// TIA Portal V15.1 export
// export: Created 2020-06-12T07:35:47.5693359Z, ExportSetting None, DisplayName Totally Integrated Automation Portal, DisplayVersion V15.1, DisplayName TIA Portal Openness, DisplayVersion V15.1, DisplayName STEP 7 Professional, DisplayVersion V15.1, DisplayName STEP 7 Safety, DisplayVersion V15.1, DisplayName WinCC Advanced, DisplayVersion V15.1
FUNCTION "DED_Fan" : Void   // FC553, FBD
TITLE = Dedusting unit (SINK) control
{ S7_Optimized_Access := 'TRUE' }
// stored: SetENOAutomatically True
   VAR_TEMP
      tRelSpeed : Real;
      tFanSpeedMin : Real;
      tFanSpeedMax : Real;
      tActPress : Real;
      tClock : Bool;
      tDoSchake : Bool;
      tSpdContLock : Bool;
      tSetPress : Real;
   END_VAR
BEGIN

REGION Network 1: AX1LD3.M01: Fan
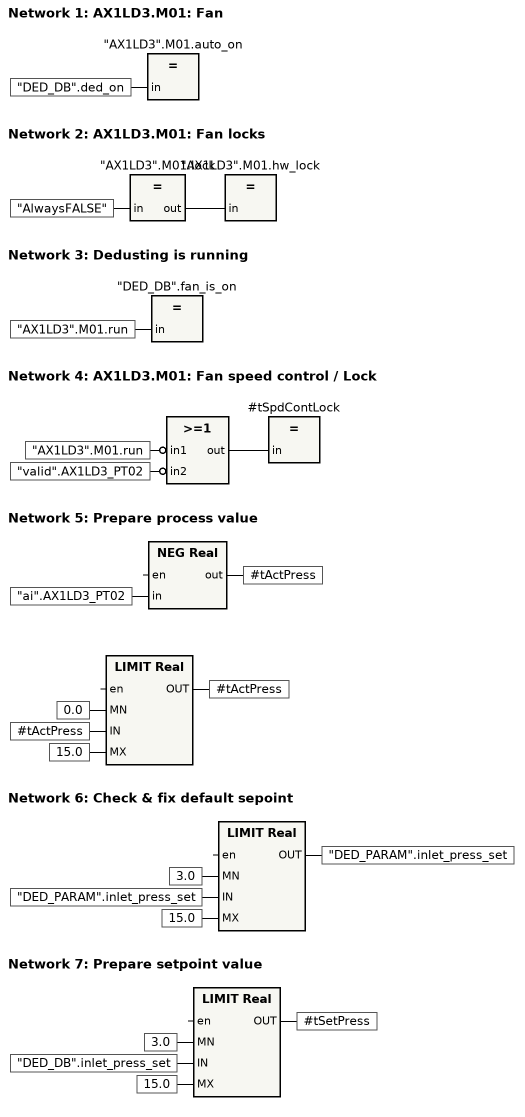
   "AX1LD3".M01.auto_on := "DED_DB".ded_on;
END_REGION

REGION Network 2: AX1LD3.M01: Fan locks
   "AX1LD3".M01.lock := "AlwaysFALSE";
   "AX1LD3".M01.hw_lock := "AlwaysFALSE";
END_REGION

REGION Network 3: Dedusting is running
   "DED_DB".fan_is_on := "AX1LD3".M01.run;
END_REGION

REGION Network 4: AX1LD3.M01: Fan speed control / Lock
   #tSpdContLock := NOT "AX1LD3".M01.run OR NOT "valid".AX1LD3_PT02;
END_REGION

REGION Network 5: Prepare process value
   #tActPress := -"ai".AX1LD3_PT02;
   #tActPress := LIMIT(MN := 0.0, IN := #tActPress, MX := 15.0);
END_REGION

REGION Network 6: Check & fix default sepoint
   "DED_PARAM".inlet_press_set := LIMIT(MN := 3.0, IN := "DED_PARAM".inlet_press_set, MX := 15.0);
END_REGION

REGION Network 7: Prepare setpoint value
   #tSetPress := LIMIT(MN := 3.0, IN := "DED_DB".inlet_press_set, MX := 15.0);
END_REGION

REGION Network 8: AX1LD3.M01: Fan speed control
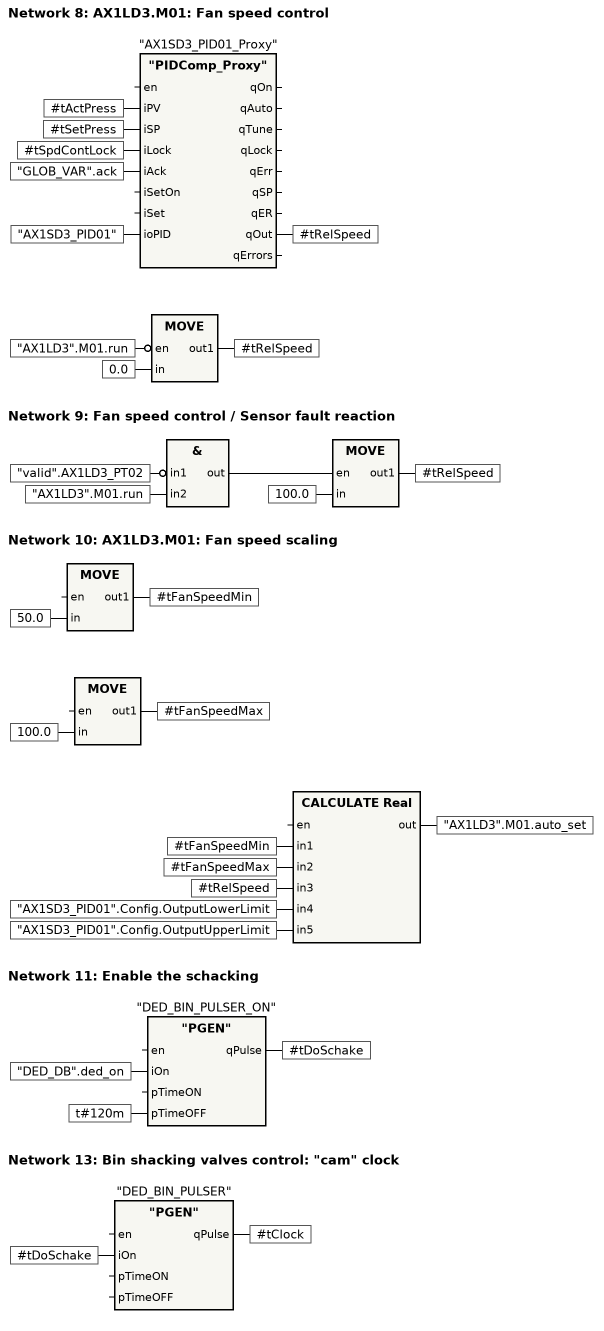
   "AX1SD3_PID01_Proxy"(iPV := #tActPress,   // "PIDComp_Proxy"
                        iSP := #tSetPress,
                        iLock := #tSpdContLock,
                        iAck := "GLOB_VAR".ack,
                        ioPID := "AX1SD3_PID01",
                        qOut => #tRelSpeed);
   IF NOT "AX1LD3".M01.run THEN #tRelSpeed := 0.0; END_IF;
END_REGION

REGION Network 9: Fan speed control / Sensor fault reaction
   IF NOT "valid".AX1LD3_PT02 AND "AX1LD3".M01.run THEN #tRelSpeed := 100.0; END_IF;
END_REGION

REGION Network 10: AX1LD3.M01: Fan speed scaling
   #tFanSpeedMin := 50.0;
   #tFanSpeedMax := 100.0;
   "AX1LD3".M01.auto_set := #tFanSpeedMin + (#tFanSpeedMax - #tFanSpeedMin) * ((#tRelSpeed - "AX1SD3_PID01".Config.OutputLowerLimit) / ("AX1SD3_PID01".Config.OutputUpperLimit - "AX1SD3_PID01".Config.OutputLowerLimit));
END_REGION

REGION Network 11: Enable the schacking
   // WARNING! DO NOT LINK THE pTimeON
   "DED_BIN_PULSER_ON"(iOn := "DED_DB".ded_on, pTimeOFF := t#120m, qPulse => #tDoSchake);   // "PGEN"
END_REGION

REGION Network 12 (SCL): Calculate time for activated stated
   "DED_BIN_PULSER_ON".pTimeON := 4 * ("DED_BIN_PULSER".pTimeOFF + "DED_BIN_PULSER".pTimeON);
END_REGION

REGION Network 13: Bin shacking valves control: "cam" clock
   "DED_BIN_PULSER"(iOn := #tDoSchake, qPulse => #tClock);   // "PGEN"
END_REGION

REGION Network 14: Bin shacking valves control
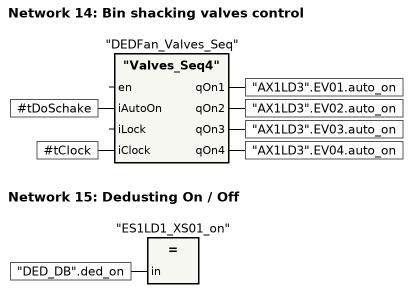
   "DEDFan_Valves_Seq"(iAutoOn := #tDoSchake,   // "Valves_Seq4"
                       iClock := #tClock,
                       qOn1 => "AX1LD3".EV01.auto_on,
                       qOn2 => "AX1LD3".EV02.auto_on,
                       qOn3 => "AX1LD3".EV03.auto_on,
                       qOn4 => "AX1LD3".EV04.auto_on);
END_REGION

REGION Network 15: Dedusting On / Off
   // TODO: clarify the meaning of signal
   "ES1LD1_XS01_on" := "DED_DB".ded_on;
END_REGION
END_FUNCTION
